GLOBALCONSTANTS myComputers (* Global constants *)
  (* Standard: 61499-1; Description: Copyright (c) 2023 HR Agrartechnik GmbH This program and the accompanying materials are made available under the terms of the Eclipse Public License 2.0 which is available at https://www.eclipse.org/legal/epl-2.0/ SPDX-License-Identifier: EPL-2.0 *)
  (* Version 1.0, 2023-10-22, Franz Höpfinger, HR Agrartechnik GmbH *)
  VAR_GLOBAL CONSTANT
    C_PC_A : WSTRING := "192.168.178.60:61499";
    C_PC_B : WSTRING := "192.168.178.62:61499";
  END_VAR
END_GLOBALCONSTANTS
